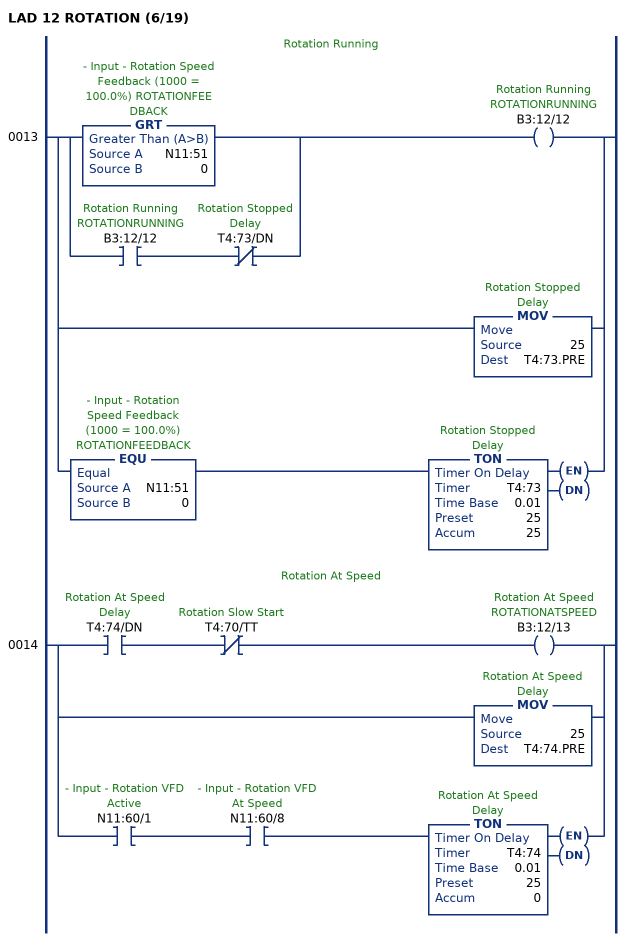
% Rung: 13 %
% Rotation Running %
SOR BST BST GRT N11:51 0 NXB XIC B3:12/12 XIO T4:73/DN BND OTE B3:12/12 NXB MOV 25 T4:73.PRE NXB EQU N11:51 0 TON T4:73 0.01 25 25 BND EOR
%   N11:51  ROTATIONFEEDBACK  "- Input - Rotation Speed Feedback (1000 = 100.0%)" %
%   B3:12/12  ROTATIONRUNNING  "Rotation Running" %
%   T4:73  "Rotation Stopped Delay" %
% Rung: 14 %
% Rotation At Speed %
SOR BST XIC T4:74/DN XIO T4:70/TT OTE B3:12/13 NXB MOV 25 T4:74.PRE NXB XIC N11:60/1 XIC N11:60/8 TON T4:74 0.01 25 0 BND EOR
%   T4:74  "Rotation At Speed Delay" %
%   T4:70  "Rotation Slow Start" %
%   B3:12/13  ROTATIONATSPEED  "Rotation At Speed" %
%   N11:60/1  "- Input - Rotation VFD Active" %
%   N11:60/8  "- Input - Rotation VFD At Speed" %

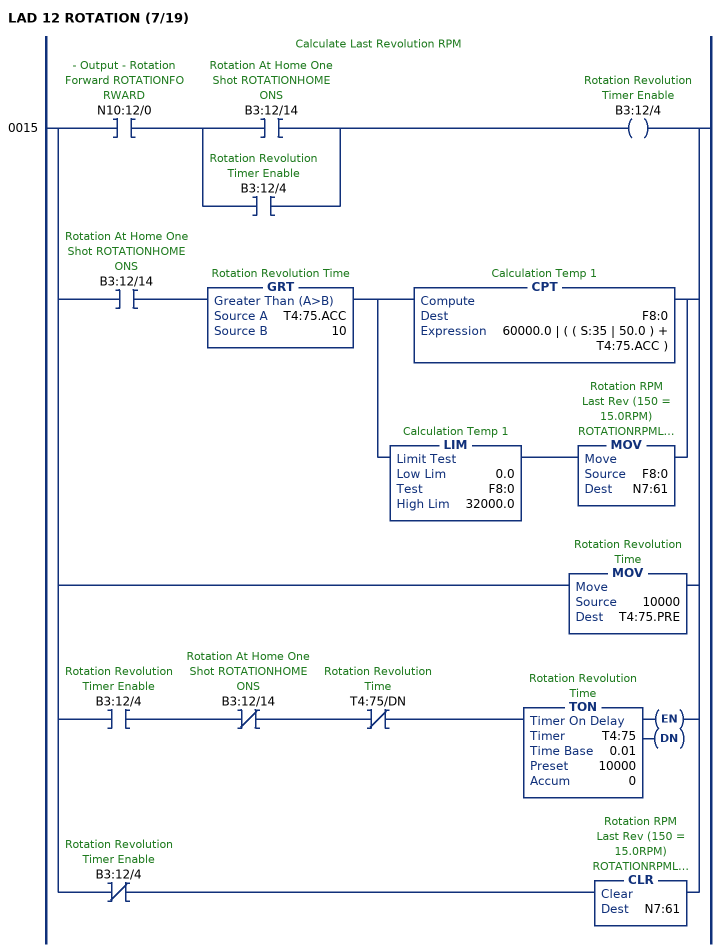
% Rung: 15 %
% Calculate Last Revolution RPM %
SOR BST XIC N10:12/0 BST XIC B3:12/14 NXB XIC B3:12/4 BND OTE B3:12/4 NXB XIC B3:12/14 GRT T4:75.ACC 10 BST CPT F8:0 " 60000.0 | ( ( S:35 | 50.0 ) + T4:75.ACC ) " NXB LIM 0.0 F8:0 32000.0 MOV F8:0 N7:61 BND NXB MOV 10000 T4:75.PRE NXB XIC B3:12/4 XIO B3:12/14 XIO T4:75/DN TON T4:75 0.01 10000 0 NXB XIO B3:12/4 CLR N7:61 BND EOR
%   N10:12/0  ROTATIONFORWARD  "- Output - Rotation Forward" %
%   B3:12/14  ROTATIONHOMEONS  "Rotation At Home One Shot" %
%   B3:12/4  "Rotation Revolution Timer Enable" %
%   T4:75  "Rotation Revolution Time" %
%   F8:0  "Calculation Temp 1" %
%   S:35  "Last 1 ms Scan Time" %
%   N7:61  ROTATIONRPMLAST  "Rotation RPM Last Rev (150 = 15.0RPM)" %

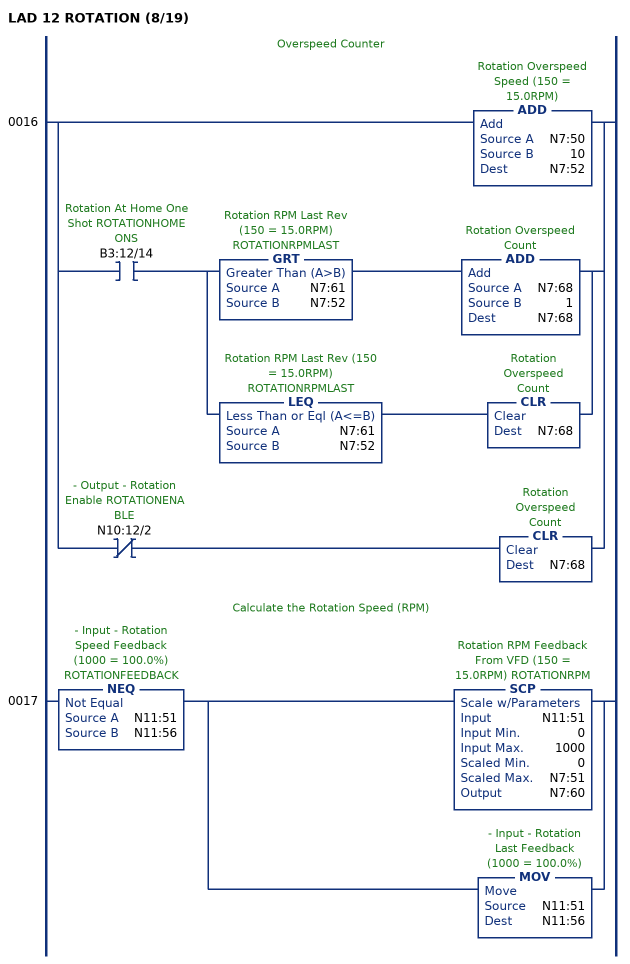
% Rung: 16 %
% Overspeed Counter %
SOR BST ADD N7:50 10 N7:52 NXB XIC B3:12/14 BST GRT N7:61 N7:52 ADD N7:68 1 N7:68 NXB LEQ N7:61 N7:52 CLR N7:68 BND NXB XIO N10:12/2 CLR N7:68 BND EOR
%   N7:50  ROTATIONBASESPEED  "Rotation Base Speed (150 = 15.0RPM)" %
%   N7:52  "Rotation Overspeed Speed (150 = 15.0RPM)" %
%   B3:12/14  ROTATIONHOMEONS  "Rotation At Home One Shot" %
%   N7:61  ROTATIONRPMLAST  "Rotation RPM Last Rev (150 = 15.0RPM)" %
%   N7:68  "Rotation Overspeed Count" %
%   N10:12/2  ROTATIONENABLE  "- Output - Rotation Enable" %
% Rung: 17 %
% Calculate the Rotation Speed (RPM) %
SOR NEQ N11:51 N11:56 BST SCP N11:51 0 1000 0 N7:51 N7:60 NXB MOV N11:51 N11:56 BND EOR
%   N11:51  ROTATIONFEEDBACK  "- Input - Rotation Speed Feedback (1000 = 100.0%)" %
%   N11:56  "- Input - Rotation Last Feedback (1000 = 100.0%)" %
%   N7:51  ROTATIONMAXSPEED  "Rotation Max Speed (150 = 15.0RPM)" %
%   N7:60  ROTATIONRPM  "Rotation RPM Feedback From VFD (150 = 15.0RPM)" %

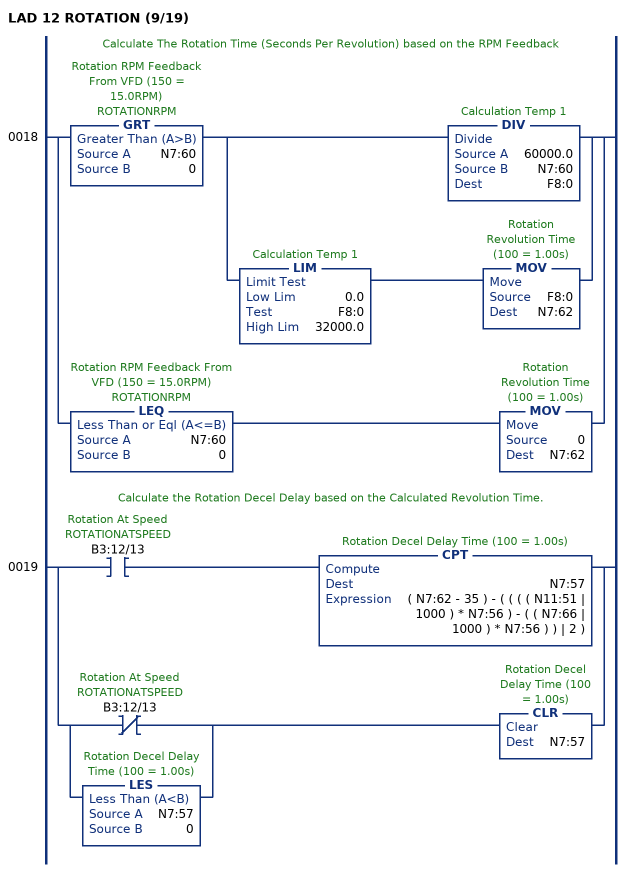
% Rung: 18 %
% Calculate The Rotation Time (Seconds Per Revolution) based on the RPM Feedback %
SOR BST GRT N7:60 0 BST DIV 60000.0 N7:60 F8:0 NXB LIM 0.0 F8:0 32000.0 MOV F8:0 N7:62 BND NXB LEQ N7:60 0 MOV 0 N7:62 BND EOR
%   N7:60  ROTATIONRPM  "Rotation RPM Feedback From VFD (150 = 15.0RPM)" %
%   F8:0  "Calculation Temp 1" %
%   N7:62  "Rotation Revolution Time (100 = 1.00s)" %
% Rung: 19 %
% Calculate the Rotation Decel Delay based on the Calculated Revolution Time. %
SOR BST XIC B3:12/13 CPT N7:57 " ( N7:62 - 35 ) - ( ( ( ( N11:51 | 1000 ) * N7:56 ) - ( ( N7:66 | 1000 ) * N7:56 ) ) | 2 ) " NXB BST XIO B3:12/13 NXB LES N7:57 0 BND CLR N7:57 BND EOR
%   B3:12/13  ROTATIONATSPEED  "Rotation At Speed" %
%   N7:57  "Rotation Decel Delay Time (100 = 1.00s)" %
%   N7:62  "Rotation Revolution Time (100 = 1.00s)" %
%   N11:51  ROTATIONFEEDBACK  "- Input - Rotation Speed Feedback (1000 = 100.0%)" %
%   N7:56  "Rotation Decel Time (100 = 1.00s)" %
%   N7:66  "Rotation Home Speed (25 = 2.5RPM)" %

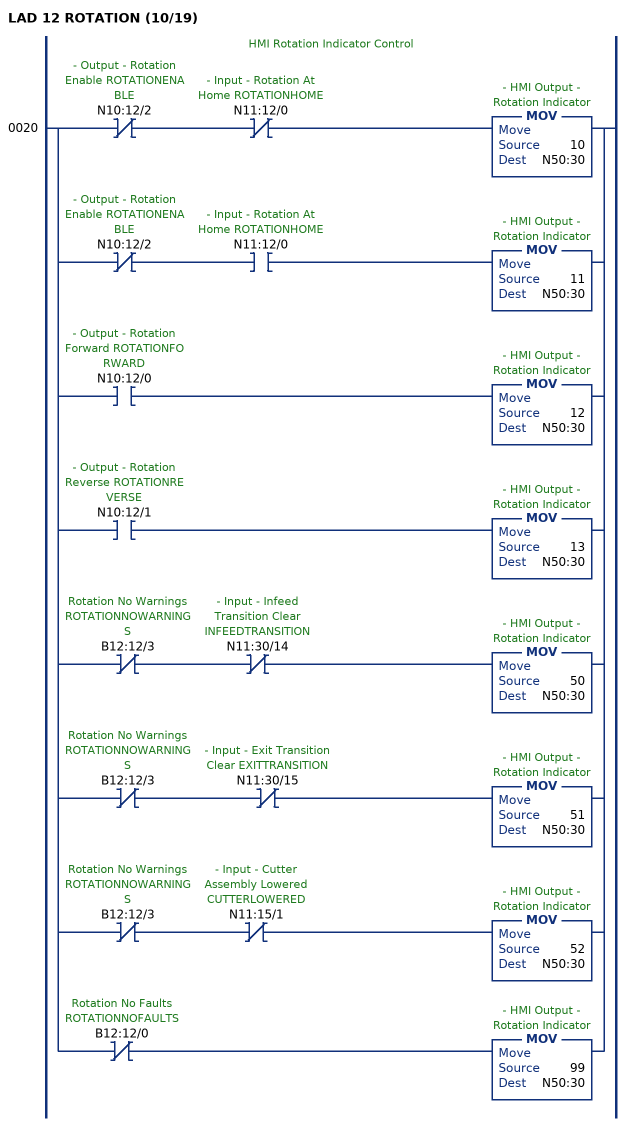
% Rung: 20 %
% HMI Rotation Indicator Control %
SOR BST XIO N10:12/2 XIO N11:12/0 MOV 10 N50:30 NXB XIO N10:12/2 XIC N11:12/0 MOV 11 N50:30 NXB XIC N10:12/0 MOV 12 N50:30 NXB XIC N10:12/1 MOV 13 N50:30 NXB XIO B12:12/3 XIO N11:30/14 MOV 50 N50:30 NXB XIO B12:12/3 XIO N11:30/15 MOV 51 N50:30 NXB XIO B12:12/3 XIO N11:15/1 MOV 52 N50:30 NXB XIO B12:12/0 MOV 99 N50:30 BND EOR
%   N10:12/2  ROTATIONENABLE  "- Output - Rotation Enable" %
%   N11:12/0  ROTATIONHOME  "- Input - Rotation At Home" %
%   N50:30  "- HMI Output - Rotation Indicator" %
%   N10:12/0  ROTATIONFORWARD  "- Output - Rotation Forward" %
%   N10:12/1  ROTATIONREVERSE  "- Output - Rotation Reverse" %
%   B12:12/3  ROTATIONNOWARNINGS  "Rotation No Warnings" %
%   N11:30/14  INFEEDTRANSITION  "- Input - Infeed Transition Clear" %
%   N11:30/15  EXITTRANSITION  "- Input - Exit Transition Clear" %
%   N11:15/1  CUTTERLOWERED  "- Input - Cutter Assembly Lowered" %
%   B12:12/0  ROTATIONNOFAULTS  "Rotation No Faults" %

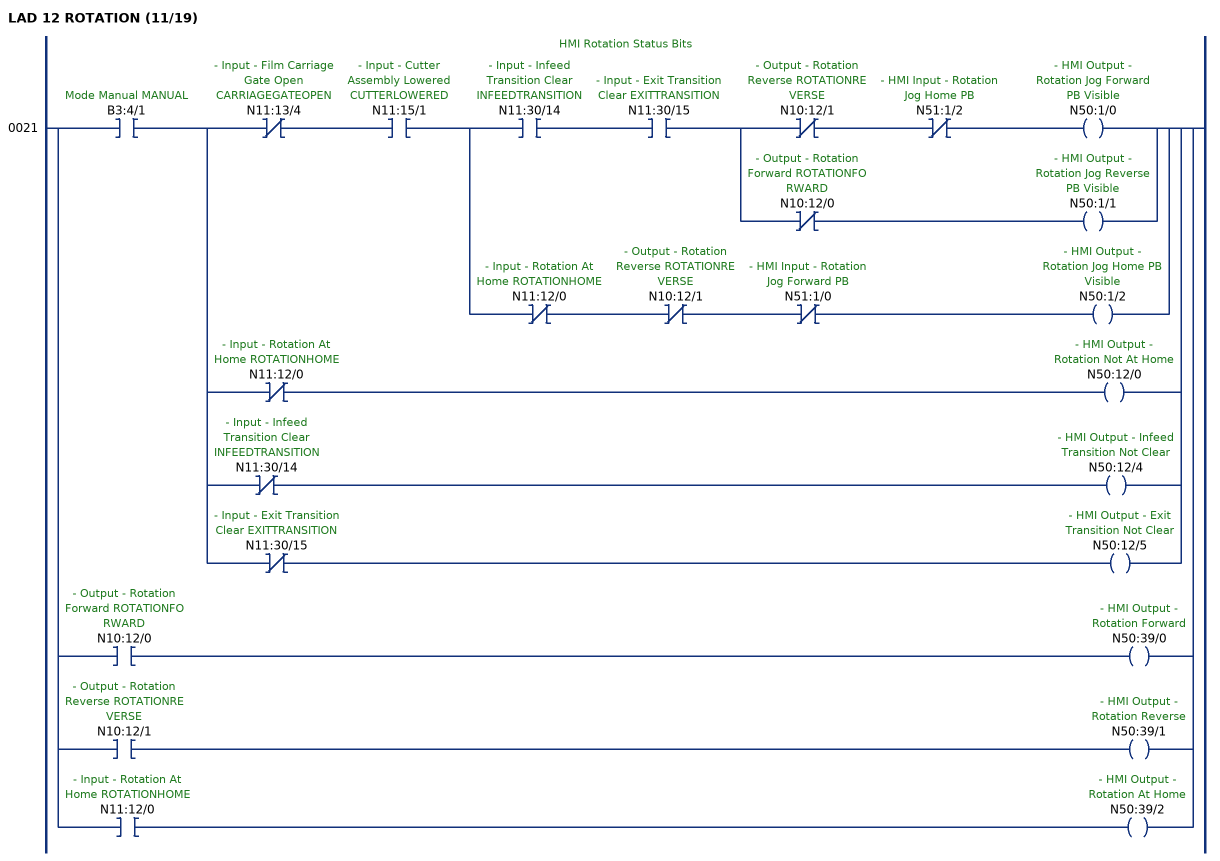
% Rung: 21 %
% HMI Rotation Status Bits %
SOR BST XIC B3:4/1 BST XIO N11:13/4 XIC N11:15/1 BST XIC N11:30/14 XIC N11:30/15 BST XIO N10:12/1 XIO N51:1/2 OTE N50:1/0 NXB XIO N10:12/0 OTE N50:1/1 BND NXB XIO N11:12/0 XIO N10:12/1 XIO N51:1/0 OTE N50:1/2 BND NXB XIO N11:12/0 OTE N50:12/0 NXB XIO N11:30/14 OTE N50:12/4 NXB XIO N11:30/15 OTE N50:12/5 BND NXB XIC N10:12/0 OTE N50:39/0 NXB XIC N10:12/1 OTE N50:39/1 NXB XIC N11:12/0 OTE N50:39/2 BND EOR
%   B3:4/1  MANUAL  "Mode Manual" %
%   N11:13/4  CARRIAGEGATEOPEN  "- Input - Film Carriage Gate Open" %
%   N11:15/1  CUTTERLOWERED  "- Input - Cutter Assembly Lowered" %
%   N11:30/14  INFEEDTRANSITION  "- Input - Infeed Transition Clear" %
%   N11:30/15  EXITTRANSITION  "- Input - Exit Transition Clear" %
%   N10:12/1  ROTATIONREVERSE  "- Output - Rotation Reverse" %
%   N51:1/2  "- HMI Input - Rotation Jog Home PB" %
%   N50:1/0  "- HMI Output - Rotation Jog Forward PB Visible" %
%   N10:12/0  ROTATIONFORWARD  "- Output - Rotation Forward" %
%   N50:1/1  "- HMI Output - Rotation Jog Reverse PB Visible" %
%   N11:12/0  ROTATIONHOME  "- Input - Rotation At Home" %
%   N51:1/0  "- HMI Input - Rotation Jog Forward PB" %
%   N50:1/2  "- HMI Output - Rotation Jog Home PB Visible" %
%   N50:12/0  "- HMI Output - Rotation Not At Home" %
%   N50:12/4  "- HMI Output - Infeed Transition Not Clear" %
%   N50:12/5  "- HMI Output - Exit Transition Not Clear" %
%   N50:39/0  "- HMI Output - Rotation Forward" %
%   N50:39/1  "- HMI Output - Rotation Reverse" %
%   N50:39/2  "- HMI Output - Rotation At Home" %

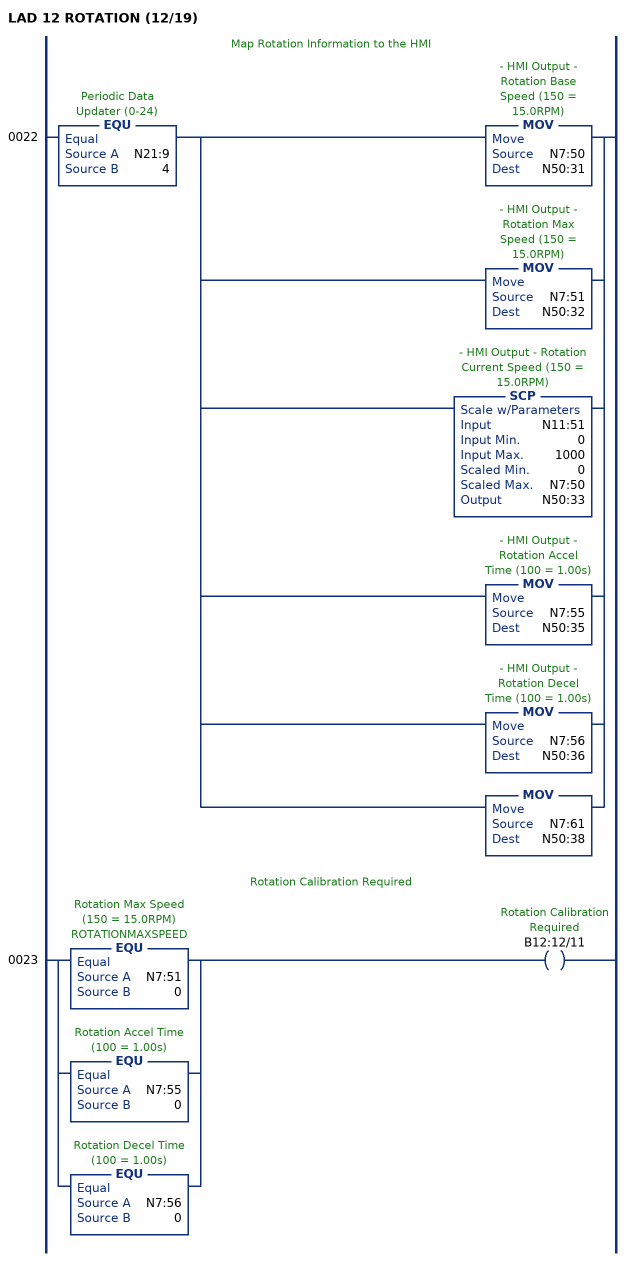
% Rung: 22 %
% Map Rotation Information to the HMI %
SOR EQU N21:9 4 BST MOV N7:50 N50:31 NXB MOV N7:51 N50:32 NXB SCP N11:51 0 1000 0 N7:50 N50:33 NXB MOV N7:55 N50:35 NXB MOV N7:56 N50:36 NXB MOV N7:61 N50:38 BND EOR
%   N21:9  "Periodic Data Updater (0-24)" %
%   N7:50  ROTATIONBASESPEED  "Rotation Base Speed (150 = 15.0RPM)" %
%   N50:31  "- HMI Output - Rotation Base Speed (150 = 15.0RPM)" %
%   N7:51  ROTATIONMAXSPEED  "Rotation Max Speed (150 = 15.0RPM)" %
%   N50:32  "- HMI Output - Rotation Max Speed (150 = 15.0RPM)" %
%   N11:51  ROTATIONFEEDBACK  "- Input - Rotation Speed Feedback (1000 = 100.0%)" %
%   N50:33  "- HMI Output - Rotation Current Speed (150 = 15.0RPM)" %
%   N7:55  "Rotation Accel Time (100 = 1.00s)" %
%   N50:35  "- HMI Output - Rotation Accel Time (100 = 1.00s)" %
%   N7:56  "Rotation Decel Time (100 = 1.00s)" %
%   N50:36  "- HMI Output - Rotation Decel Time (100 = 1.00s)" %
%   N7:61  ROTATIONRPMLAST  "Rotation RPM Last Rev (150 = 15.0RPM)" %
% Rung: 23 %
% Rotation Calibration Required %
SOR BST EQU N7:51 0 NXB EQU N7:55 0 NXB EQU N7:56 0 BND OTE B12:12/11 EOR
%   N7:51  ROTATIONMAXSPEED  "Rotation Max Speed (150 = 15.0RPM)" %
%   N7:55  "Rotation Accel Time (100 = 1.00s)" %
%   N7:56  "Rotation Decel Time (100 = 1.00s)" %
%   B12:12/11  "Rotation Calibration Required" %

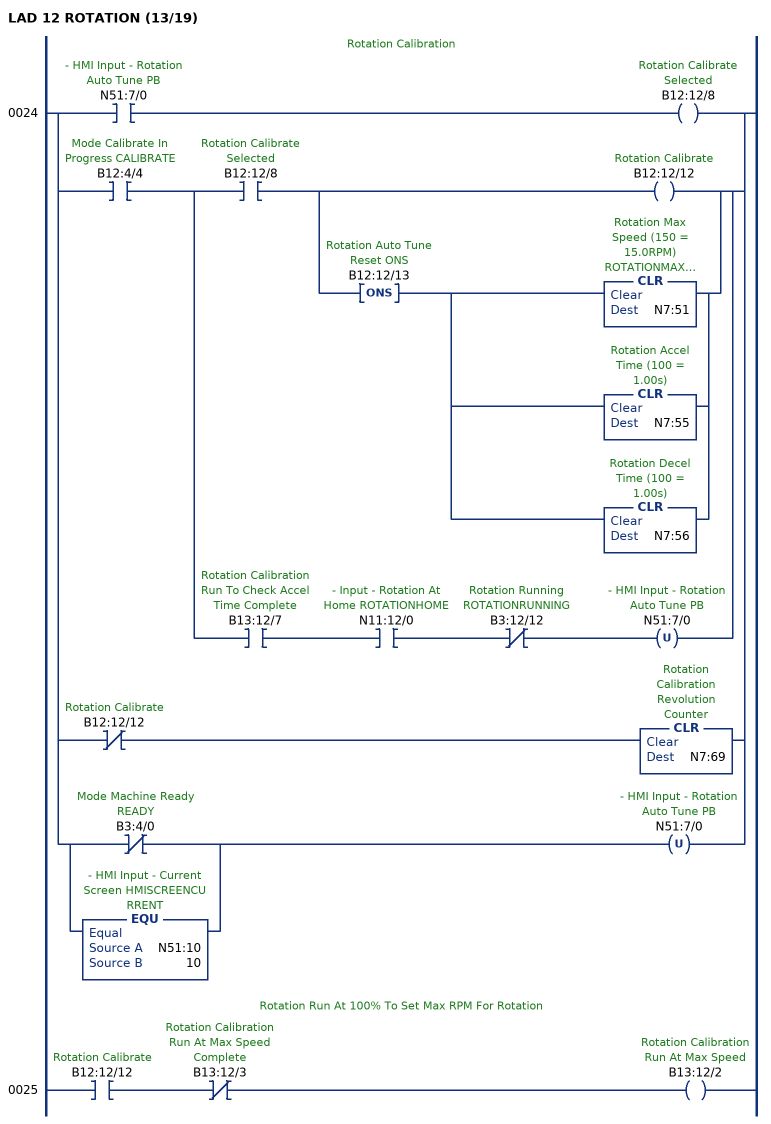
% Rung: 24 %
% Rotation Calibration %
SOR BST XIC N51:7/0 OTE B12:12/8 NXB XIC B12:4/4 BST XIC B12:12/8 BST OTE B12:12/12 NXB ONS B12:12/13 BST CLR N7:51 NXB CLR N7:55 NXB CLR N7:56 BND BND NXB XIC B13:12/7 XIC N11:12/0 XIO B3:12/12 OTU N51:7/0 BND NXB XIO B12:12/12 CLR N7:69 NXB BST XIO B3:4/0 NXB EQU N51:10 10 BND OTU N51:7/0 BND EOR
%   N51:7/0  "- HMI Input - Rotation Auto Tune PB" %
%   B12:12/8  "Rotation Calibrate Selected" %
%   B12:4/4  CALIBRATE  "Mode Calibrate In Progress" %
%   B12:12/12  "Rotation Calibrate" %
%   B12:12/13  "Rotation Auto Tune Reset ONS" %
%   N7:51  ROTATIONMAXSPEED  "Rotation Max Speed (150 = 15.0RPM)" %
%   N7:55  "Rotation Accel Time (100 = 1.00s)" %
%   N7:56  "Rotation Decel Time (100 = 1.00s)" %
%   B13:12/7  "Rotation Calibration Run To Check Accel Time Complete" %
%   N11:12/0  ROTATIONHOME  "- Input - Rotation At Home" %
%   B3:12/12  ROTATIONRUNNING  "Rotation Running" %
%   N7:69  "Rotation Calibration Revolution Counter" %
%   B3:4/0  READY  "Mode Machine Ready" %
%   N51:10  HMISCREENCURRENT  "- HMI Input - Current Screen" %
% Rung: 25 %
% Rotation Run At 100% To Set Max RPM For Rotation %
SOR XIC B12:12/12 XIO B13:12/3 OTE B13:12/2 EOR
%   B12:12/12  "Rotation Calibrate" %
%   B13:12/3  "Rotation Calibration Run At Max Speed Complete" %
%   B13:12/2  "Rotation Calibration Run At Max Speed" %

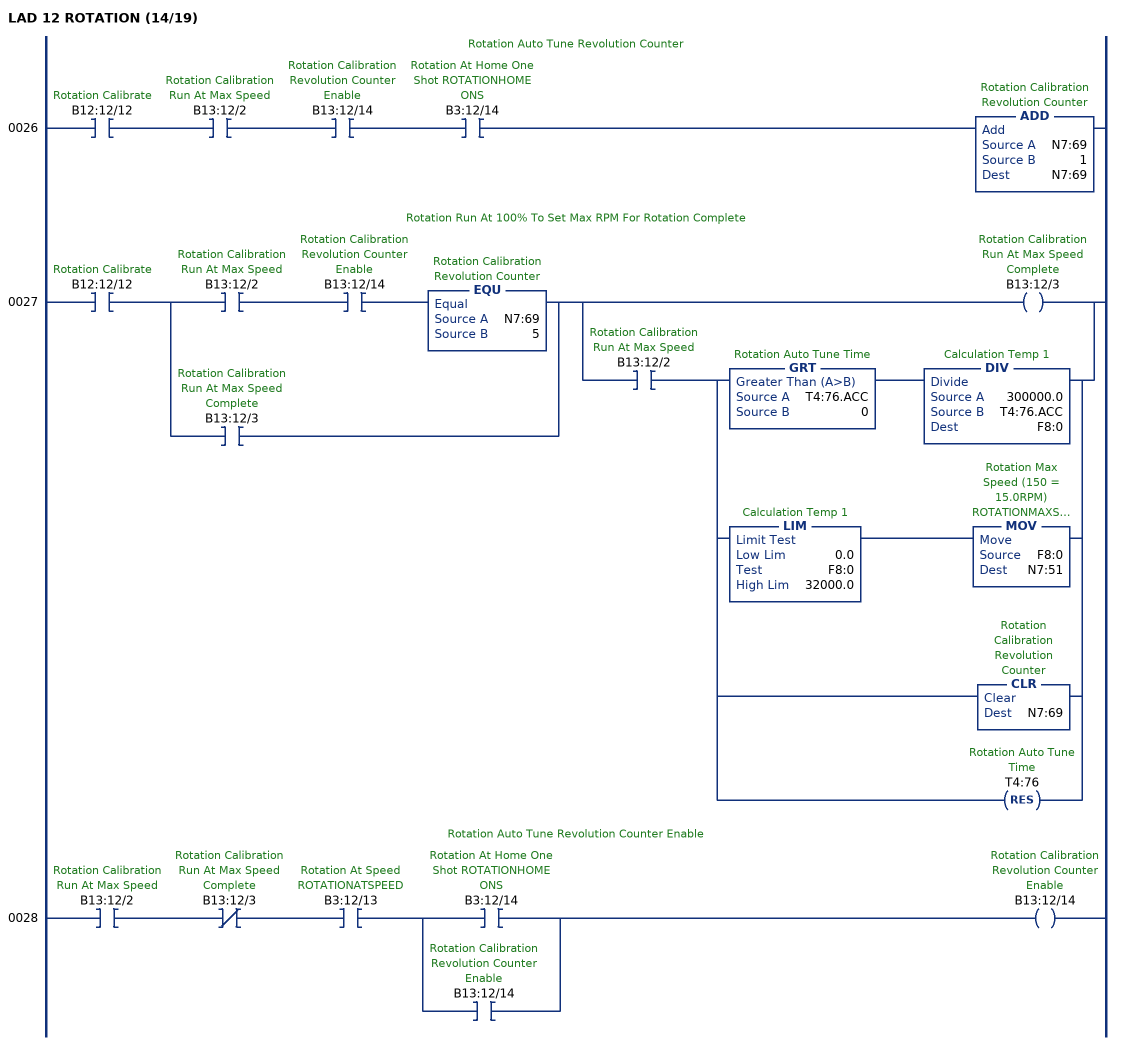
% Rung: 26 %
% Rotation Auto Tune Revolution Counter %
SOR XIC B12:12/12 XIC B13:12/2 XIC B13:12/14 XIC B3:12/14 ADD N7:69 1 N7:69 EOR
%   B12:12/12  "Rotation Calibrate" %
%   B13:12/2  "Rotation Calibration Run At Max Speed" %
%   B13:12/14  "Rotation Calibration Revolution Counter Enable" %
%   B3:12/14  ROTATIONHOMEONS  "Rotation At Home One Shot" %
%   N7:69  "Rotation Calibration Revolution Counter" %
% Rung: 27 %
% Rotation Run At 100% To Set Max RPM For Rotation Complete %
SOR XIC B12:12/12 BST XIC B13:12/2 XIC B13:12/14 EQU N7:69 5 NXB XIC B13:12/3 BND BST OTE B13:12/3 NXB XIC B13:12/2 BST GRT T4:76.ACC 0 DIV 300000.0 T4:76.ACC F8:0 NXB LIM 0.0 F8:0 32000.0 MOV F8:0 N7:51 NXB CLR N7:69 NXB RES T4:76 BND BND EOR
%   B12:12/12  "Rotation Calibrate" %
%   B13:12/2  "Rotation Calibration Run At Max Speed" %
%   B13:12/14  "Rotation Calibration Revolution Counter Enable" %
%   N7:69  "Rotation Calibration Revolution Counter" %
%   B13:12/3  "Rotation Calibration Run At Max Speed Complete" %
%   T4:76  "Rotation Auto Tune Time" %
%   F8:0  "Calculation Temp 1" %
%   N7:51  ROTATIONMAXSPEED  "Rotation Max Speed (150 = 15.0RPM)" %
% Rung: 28 %
% Rotation Auto Tune Revolution Counter Enable %
SOR XIC B13:12/2 XIO B13:12/3 XIC B3:12/13 BST XIC B3:12/14 NXB XIC B13:12/14 BND OTE B13:12/14 EOR
%   B13:12/2  "Rotation Calibration Run At Max Speed" %
%   B13:12/3  "Rotation Calibration Run At Max Speed Complete" %
%   B3:12/13  ROTATIONATSPEED  "Rotation At Speed" %
%   B3:12/14  ROTATIONHOMEONS  "Rotation At Home One Shot" %
%   B13:12/14  "Rotation Calibration Revolution Counter Enable" %

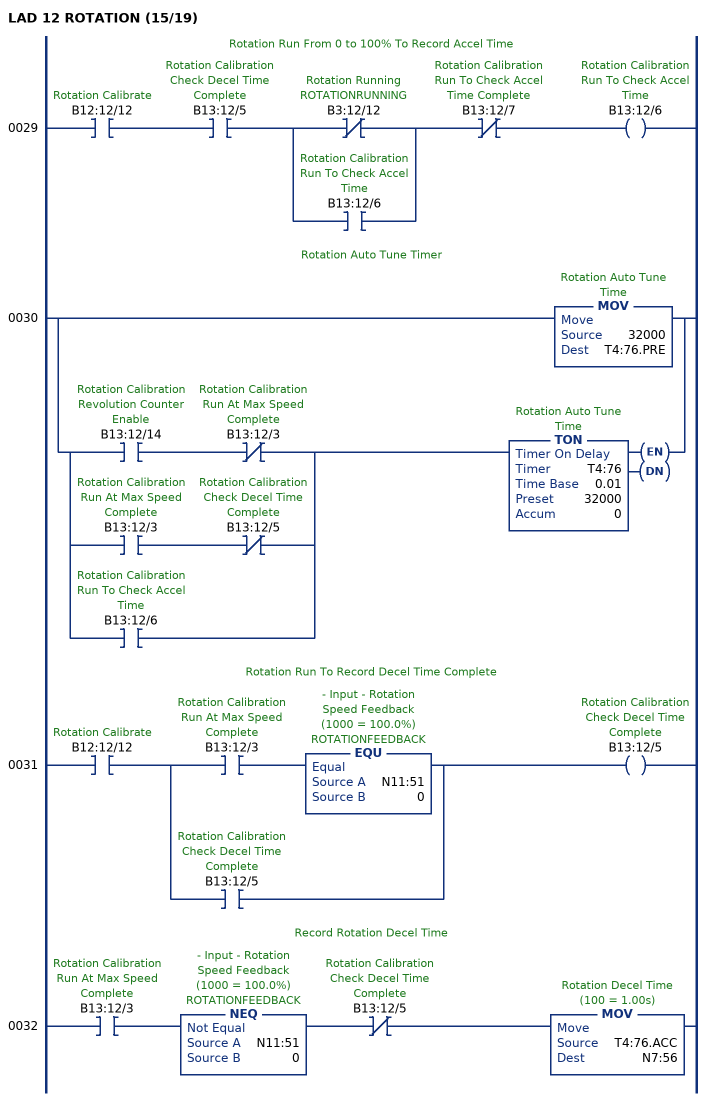
% Rung: 29 %
% Rotation Run From 0 to 100% To Record Accel Time %
SOR XIC B12:12/12 XIC B13:12/5 BST XIO B3:12/12 NXB XIC B13:12/6 BND XIO B13:12/7 OTE B13:12/6 EOR
%   B12:12/12  "Rotation Calibrate" %
%   B13:12/5  "Rotation Calibration Check Decel Time Complete" %
%   B3:12/12  ROTATIONRUNNING  "Rotation Running" %
%   B13:12/6  "Rotation Calibration Run To Check Accel Time" %
%   B13:12/7  "Rotation Calibration Run To Check Accel Time Complete" %
% Rung: 30 %
% Rotation Auto Tune Timer %
SOR BST MOV 32000 T4:76.PRE NXB BST XIC B13:12/14 XIO B13:12/3 NXB XIC B13:12/3 XIO B13:12/5 NXB XIC B13:12/6 BND TON T4:76 0.01 32000 0 BND EOR
%   T4:76  "Rotation Auto Tune Time" %
%   B13:12/14  "Rotation Calibration Revolution Counter Enable" %
%   B13:12/3  "Rotation Calibration Run At Max Speed Complete" %
%   B13:12/5  "Rotation Calibration Check Decel Time Complete" %
%   B13:12/6  "Rotation Calibration Run To Check Accel Time" %
% Rung: 31 %
% Rotation Run To Record Decel Time Complete %
SOR XIC B12:12/12 BST XIC B13:12/3 EQU N11:51 0 NXB XIC B13:12/5 BND OTE B13:12/5 EOR
%   B12:12/12  "Rotation Calibrate" %
%   B13:12/3  "Rotation Calibration Run At Max Speed Complete" %
%   N11:51  ROTATIONFEEDBACK  "- Input - Rotation Speed Feedback (1000 = 100.0%)" %
%   B13:12/5  "Rotation Calibration Check Decel Time Complete" %
% Rung: 32 %
% Record Rotation Decel Time %
SOR XIC B13:12/3 NEQ N11:51 0 XIO B13:12/5 MOV T4:76.ACC N7:56 EOR
%   B13:12/3  "Rotation Calibration Run At Max Speed Complete" %
%   N11:51  ROTATIONFEEDBACK  "- Input - Rotation Speed Feedback (1000 = 100.0%)" %
%   B13:12/5  "Rotation Calibration Check Decel Time Complete" %
%   T4:76  "Rotation Auto Tune Time" %
%   N7:56  "Rotation Decel Time (100 = 1.00s)" %

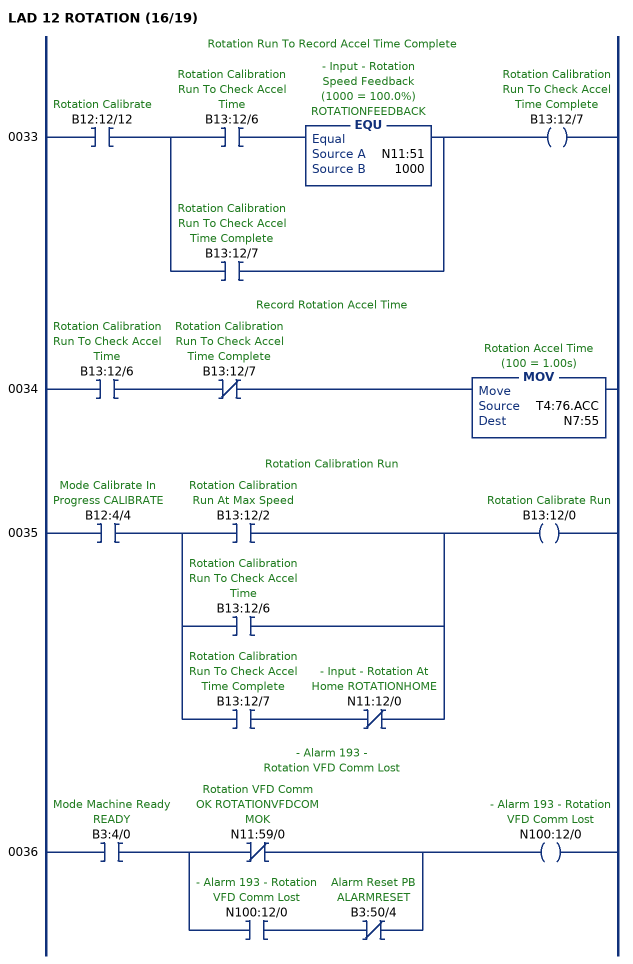
% Rung: 33 %
% Rotation Run To Record Accel Time Complete %
SOR XIC B12:12/12 BST XIC B13:12/6 EQU N11:51 1000 NXB XIC B13:12/7 BND OTE B13:12/7 EOR
%   B12:12/12  "Rotation Calibrate" %
%   B13:12/6  "Rotation Calibration Run To Check Accel Time" %
%   N11:51  ROTATIONFEEDBACK  "- Input - Rotation Speed Feedback (1000 = 100.0%)" %
%   B13:12/7  "Rotation Calibration Run To Check Accel Time Complete" %
% Rung: 34 %
% Record Rotation Accel Time %
SOR XIC B13:12/6 XIO B13:12/7 MOV T4:76.ACC N7:55 EOR
%   B13:12/6  "Rotation Calibration Run To Check Accel Time" %
%   B13:12/7  "Rotation Calibration Run To Check Accel Time Complete" %
%   T4:76  "Rotation Auto Tune Time" %
%   N7:55  "Rotation Accel Time (100 = 1.00s)" %
% Rung: 35 %
% Rotation Calibration Run %
SOR XIC B12:4/4 BST XIC B13:12/2 NXB XIC B13:12/6 NXB XIC B13:12/7 XIO N11:12/0 BND OTE B13:12/0 EOR
%   B12:4/4  CALIBRATE  "Mode Calibrate In Progress" %
%   B13:12/2  "Rotation Calibration Run At Max Speed" %
%   B13:12/6  "Rotation Calibration Run To Check Accel Time" %
%   B13:12/7  "Rotation Calibration Run To Check Accel Time Complete" %
%   N11:12/0  ROTATIONHOME  "- Input - Rotation At Home" %
%   B13:12/0  "Rotation Calibrate Run" %
% Rung: 36 %
% - Alarm 193 -
% 
% Rotation VFD Comm Lost %
SOR XIC B3:4/0 BST XIO N11:59/0 NXB XIC N100:12/0 XIO B3:50/4 BND OTE N100:12/0 EOR
%   B3:4/0  READY  "Mode Machine Ready" %
%   N11:59/0  ROTATIONVFDCOMMOK  "Rotation VFD Comm OK" %
%   N100:12/0  "- Alarm 193 - Rotation VFD Comm Lost" %
%   B3:50/4  ALARMRESET  "Alarm Reset PB" %

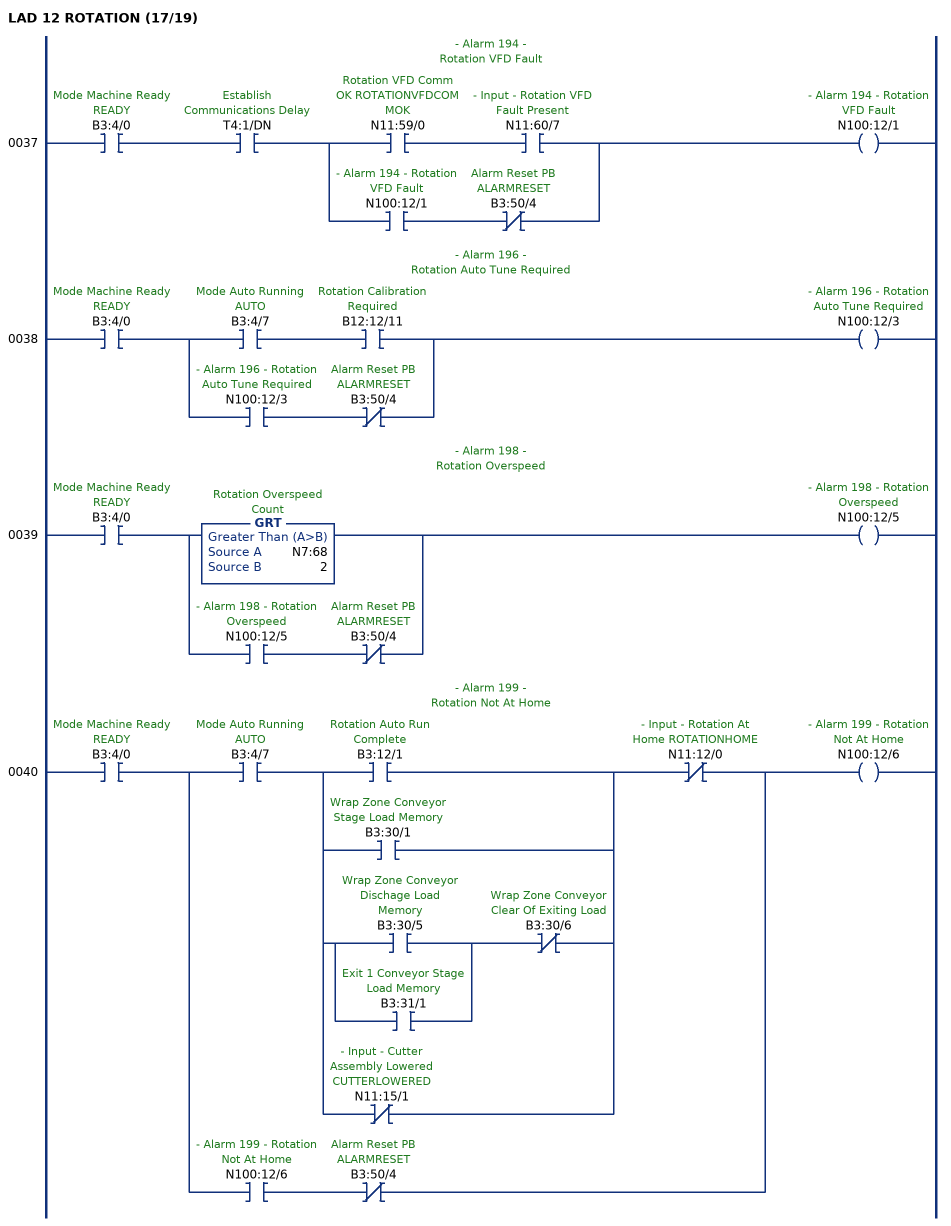
% Rung: 37 %
% - Alarm 194 -
% 
% Rotation VFD Fault %
SOR XIC B3:4/0 XIC T4:1/DN BST XIC N11:59/0 XIC N11:60/7 NXB XIC N100:12/1 XIO B3:50/4 BND OTE N100:12/1 EOR
%   B3:4/0  READY  "Mode Machine Ready" %
%   T4:1  "Establish Communications Delay" %
%   N11:59/0  ROTATIONVFDCOMMOK  "Rotation VFD Comm OK" %
%   N11:60/7  "- Input - Rotation VFD Fault Present" %
%   N100:12/1  "- Alarm 194 - Rotation VFD Fault" %
%   B3:50/4  ALARMRESET  "Alarm Reset PB" %
% Rung: 38 %
% - Alarm 196 -
% 
% Rotation Auto Tune Required %
SOR XIC B3:4/0 BST XIC B3:4/7 XIC B12:12/11 NXB XIC N100:12/3 XIO B3:50/4 BND OTE N100:12/3 EOR
%   B3:4/0  READY  "Mode Machine Ready" %
%   B3:4/7  AUTO  "Mode Auto Running" %
%   B12:12/11  "Rotation Calibration Required" %
%   N100:12/3  "- Alarm 196 - Rotation Auto Tune Required" %
%   B3:50/4  ALARMRESET  "Alarm Reset PB" %
% Rung: 39 %
% - Alarm 198 -
% 
% Rotation Overspeed %
SOR XIC B3:4/0 BST GRT N7:68 2 NXB XIC N100:12/5 XIO B3:50/4 BND OTE N100:12/5 EOR
%   B3:4/0  READY  "Mode Machine Ready" %
%   N7:68  "Rotation Overspeed Count" %
%   N100:12/5  "- Alarm 198 - Rotation Overspeed" %
%   B3:50/4  ALARMRESET  "Alarm Reset PB" %
% Rung: 40 %
% - Alarm 199 -
% 
% Rotation Not At Home %
SOR XIC B3:4/0 BST XIC B3:4/7 BST XIC B3:12/1 NXB XIC B3:30/1 NXB BST XIC B3:30/5 NXB XIC B3:31/1 BND XIO B3:30/6 NXB XIO N11:15/1 BND XIO N11:12/0 NXB XIC N100:12/6 XIO B3:50/4 BND OTE N100:12/6 EOR
%   B3:4/0  READY  "Mode Machine Ready" %
%   B3:4/7  AUTO  "Mode Auto Running" %
%   B3:12/1  "Rotation Auto Run Complete" %
%   B3:30/1  "Wrap Zone Conveyor Stage Load Memory" %
%   B3:30/5  "Wrap Zone Conveyor Dischage Load Memory" %
%   B3:31/1  "Exit 1 Conveyor Stage Load Memory" %
%   B3:30/6  "Wrap Zone Conveyor Clear Of Exiting Load" %
%   N11:15/1  CUTTERLOWERED  "- Input - Cutter Assembly Lowered" %
%   N11:12/0  ROTATIONHOME  "- Input - Rotation At Home" %
%   N100:12/6  "- Alarm 199 - Rotation Not At Home" %
%   B3:50/4  ALARMRESET  "Alarm Reset PB" %

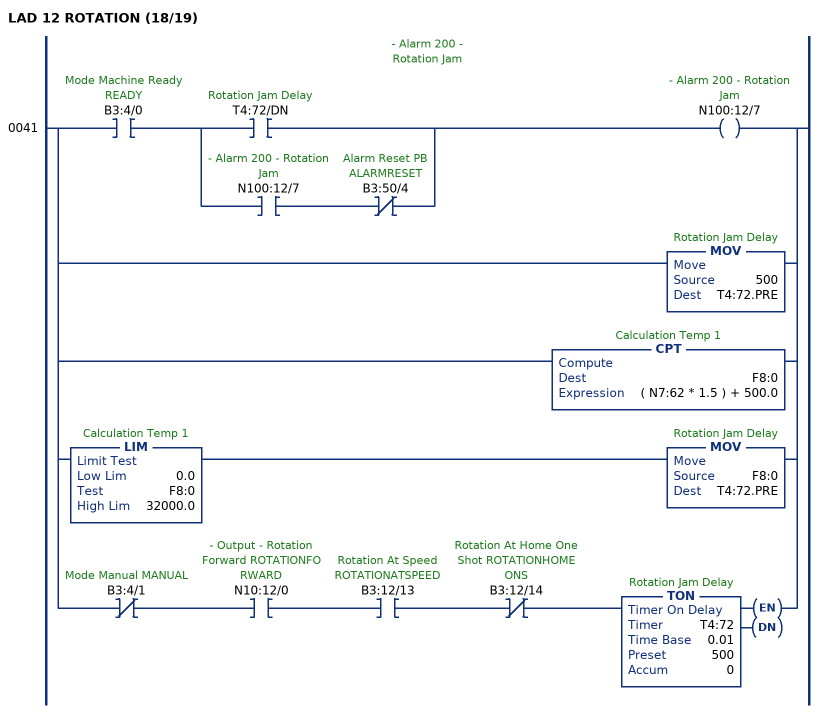
% Rung: 41 %
% - Alarm 200 -
% 
% Rotation Jam %
SOR BST XIC B3:4/0 BST XIC T4:72/DN NXB XIC N100:12/7 XIO B3:50/4 BND OTE N100:12/7 NXB BST MOV 500 T4:72.PRE NXB CPT F8:0 " ( N7:62 * 1.5 ) + 500.0 " NXB LIM 0.0 F8:0 32000.0 MOV F8:0 T4:72.PRE BND NXB XIO B3:4/1 XIC N10:12/0 XIC B3:12/13 XIO B3:12/14 TON T4:72 0.01 500 0 BND EOR
%   B3:4/0  READY  "Mode Machine Ready" %
%   T4:72  "Rotation Jam Delay" %
%   N100:12/7  "- Alarm 200 - Rotation Jam" %
%   B3:50/4  ALARMRESET  "Alarm Reset PB" %
%   F8:0  "Calculation Temp 1" %
%   N7:62  "Rotation Revolution Time (100 = 1.00s)" %
%   B3:4/1  MANUAL  "Mode Manual" %
%   N10:12/0  ROTATIONFORWARD  "- Output - Rotation Forward" %
%   B3:12/13  ROTATIONATSPEED  "Rotation At Speed" %
%   B3:12/14  ROTATIONHOMEONS  "Rotation At Home One Shot" %

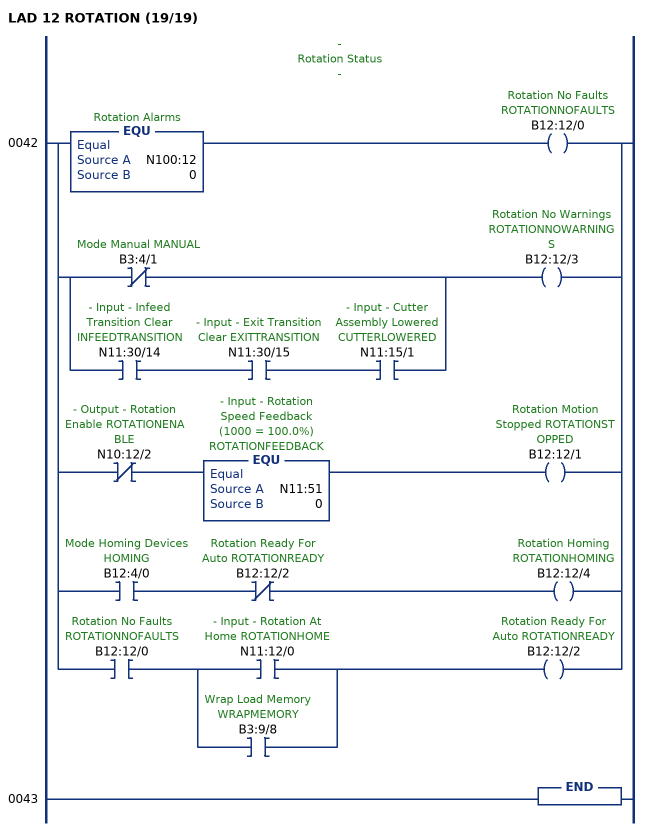
% Rung: 42 %
% -
% 
% Rotation Status
% 
% - %
SOR BST EQU N100:12 0 OTE B12:12/0 NXB BST XIO B3:4/1 NXB XIC N11:30/14 XIC N11:30/15 XIC N11:15/1 BND OTE B12:12/3 NXB XIO N10:12/2 EQU N11:51 0 OTE B12:12/1 NXB XIC B12:4/0 XIO B12:12/2 OTE B12:12/4 NXB XIC B12:12/0 BST XIC N11:12/0 NXB XIC B3:9/8 BND OTE B12:12/2 BND EOR
%   N100:12  "Rotation Alarms" %
%   B12:12/0  ROTATIONNOFAULTS  "Rotation No Faults" %
%   B3:4/1  MANUAL  "Mode Manual" %
%   N11:30/14  INFEEDTRANSITION  "- Input - Infeed Transition Clear" %
%   N11:30/15  EXITTRANSITION  "- Input - Exit Transition Clear" %
%   N11:15/1  CUTTERLOWERED  "- Input - Cutter Assembly Lowered" %
%   B12:12/3  ROTATIONNOWARNINGS  "Rotation No Warnings" %
%   N10:12/2  ROTATIONENABLE  "- Output - Rotation Enable" %
%   N11:51  ROTATIONFEEDBACK  "- Input - Rotation Speed Feedback (1000 = 100.0%)" %
%   B12:12/1  ROTATIONSTOPPED  "Rotation Motion Stopped" %
%   B12:4/0  HOMING  "Mode Homing Devices" %
%   B12:12/2  ROTATIONREADY  "Rotation Ready For Auto" %
%   B12:12/4  ROTATIONHOMING  "Rotation Homing" %
%   N11:12/0  ROTATIONHOME  "- Input - Rotation At Home" %
%   B3:9/8  WRAPMEMORY  "Wrap Load Memory" %
% Rung: 43 %
SOR END EOR

LADDER 13 "CARRIAGE"
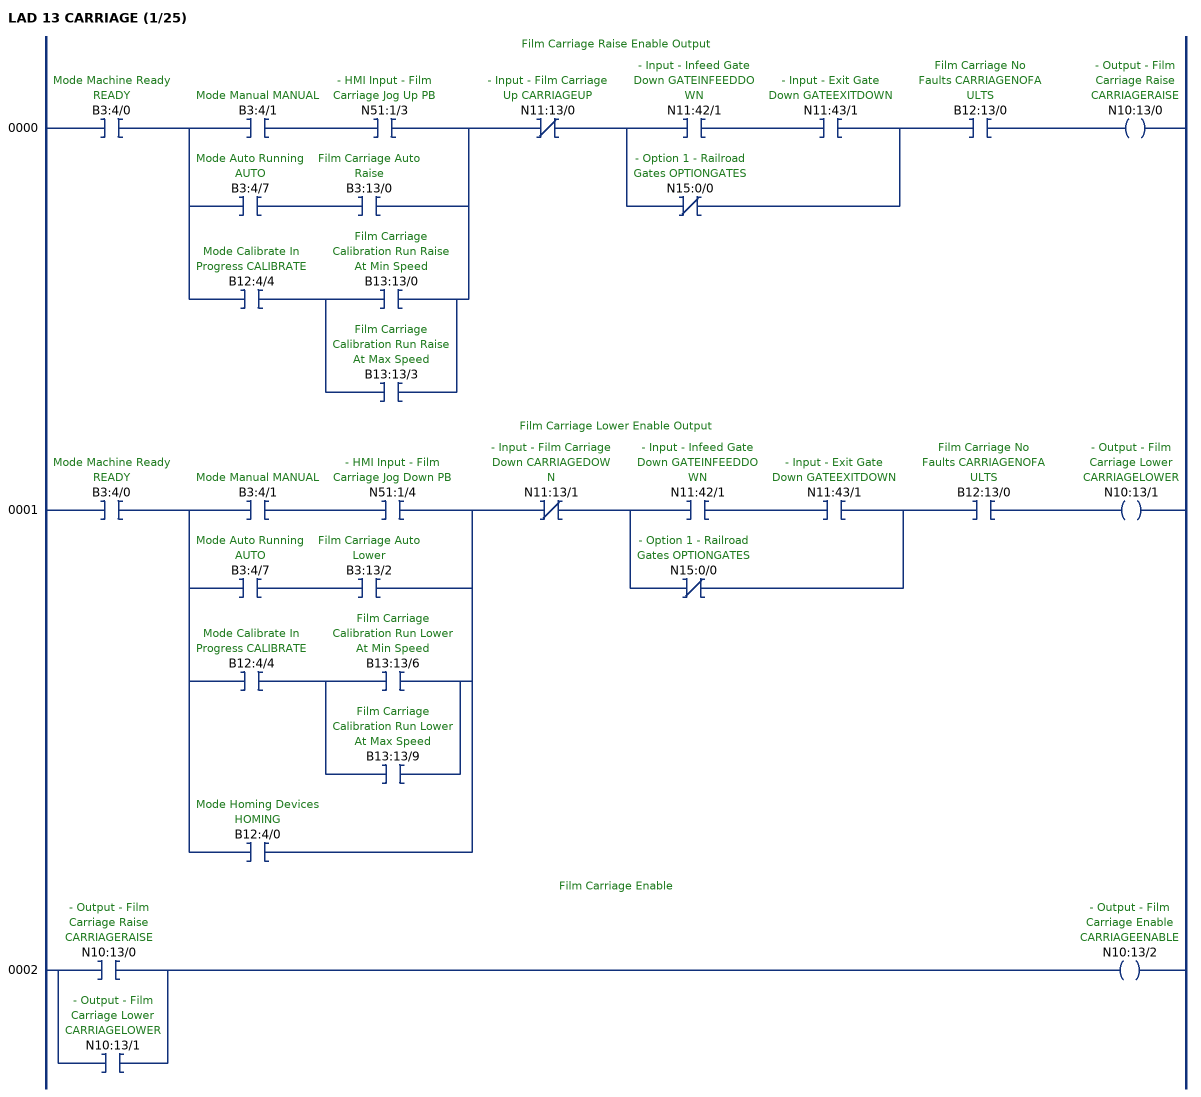
% Rung: 0 %
% Film Carriage Raise Enable Output %
SOR XIC B3:4/0 BST XIC B3:4/1 XIC N51:1/3 NXB XIC B3:4/7 XIC B3:13/0 NXB XIC B12:4/4 BST XIC B13:13/0 NXB XIC B13:13/3 BND BND XIO N11:13/0 BST XIC N11:42/1 XIC N11:43/1 NXB XIO N15:0/0 BND XIC B12:13/0 OTE N10:13/0 EOR
%   B3:4/0  READY  "Mode Machine Ready" %
%   B3:4/1  MANUAL  "Mode Manual" %
%   N51:1/3  "- HMI Input - Film Carriage Jog Up PB" %
%   B3:4/7  AUTO  "Mode Auto Running" %
%   B3:13/0  "Film Carriage Auto Raise" %
%   B12:4/4  CALIBRATE  "Mode Calibrate In Progress" %
%   B13:13/0  "Film Carriage Calibration Run Raise At Min Speed" %
%   B13:13/3  "Film Carriage Calibration Run Raise At Max Speed" %
%   N11:13/0  CARRIAGEUP  "- Input - Film Carriage Up" %
%   N11:42/1  GATEINFEEDDOWN  "- Input - Infeed Gate Down" %
%   N11:43/1  GATEEXITDOWN  "- Input - Exit Gate Down" %
%   N15:0/0  OPTIONGATES  "- Option 1 - Railroad Gates" %
%   B12:13/0  CARRIAGENOFAULTS  "Film Carriage No Faults" %
%   N10:13/0  CARRIAGERAISE  "- Output - Film Carriage Raise" %
% Rung: 1 %
% Film Carriage Lower Enable Output %
SOR XIC B3:4/0 BST XIC B3:4/1 XIC N51:1/4 NXB XIC B3:4/7 XIC B3:13/2 NXB XIC B12:4/4 BST XIC B13:13/6 NXB XIC B13:13/9 BND NXB XIC B12:4/0 BND XIO N11:13/1 BST XIC N11:42/1 XIC N11:43/1 NXB XIO N15:0/0 BND XIC B12:13/0 OTE N10:13/1 EOR
%   B3:4/0  READY  "Mode Machine Ready" %
%   B3:4/1  MANUAL  "Mode Manual" %
%   N51:1/4  "- HMI Input - Film Carriage Jog Down PB" %
%   B3:4/7  AUTO  "Mode Auto Running" %
%   B3:13/2  "Film Carriage Auto Lower" %
%   B12:4/4  CALIBRATE  "Mode Calibrate In Progress" %
%   B13:13/6  "Film Carriage Calibration Run Lower At Min Speed" %
%   B13:13/9  "Film Carriage Calibration Run Lower At Max Speed" %
%   B12:4/0  HOMING  "Mode Homing Devices" %
%   N11:13/1  CARRIAGEDOWN  "- Input - Film Carriage Down" %
%   N11:42/1  GATEINFEEDDOWN  "- Input - Infeed Gate Down" %
%   N11:43/1  GATEEXITDOWN  "- Input - Exit Gate Down" %
%   N15:0/0  OPTIONGATES  "- Option 1 - Railroad Gates" %
%   B12:13/0  CARRIAGENOFAULTS  "Film Carriage No Faults" %
%   N10:13/1  CARRIAGELOWER  "- Output - Film Carriage Lower" %
% Rung: 2 %
% Film Carriage Enable %
SOR BST XIC N10:13/0 NXB XIC N10:13/1 BND OTE N10:13/2 EOR
%   N10:13/0  CARRIAGERAISE  "- Output - Film Carriage Raise" %
%   N10:13/1  CARRIAGELOWER  "- Output - Film Carriage Lower" %
%   N10:13/2  CARRIAGEENABLE  "- Output - Film Carriage Enable" %

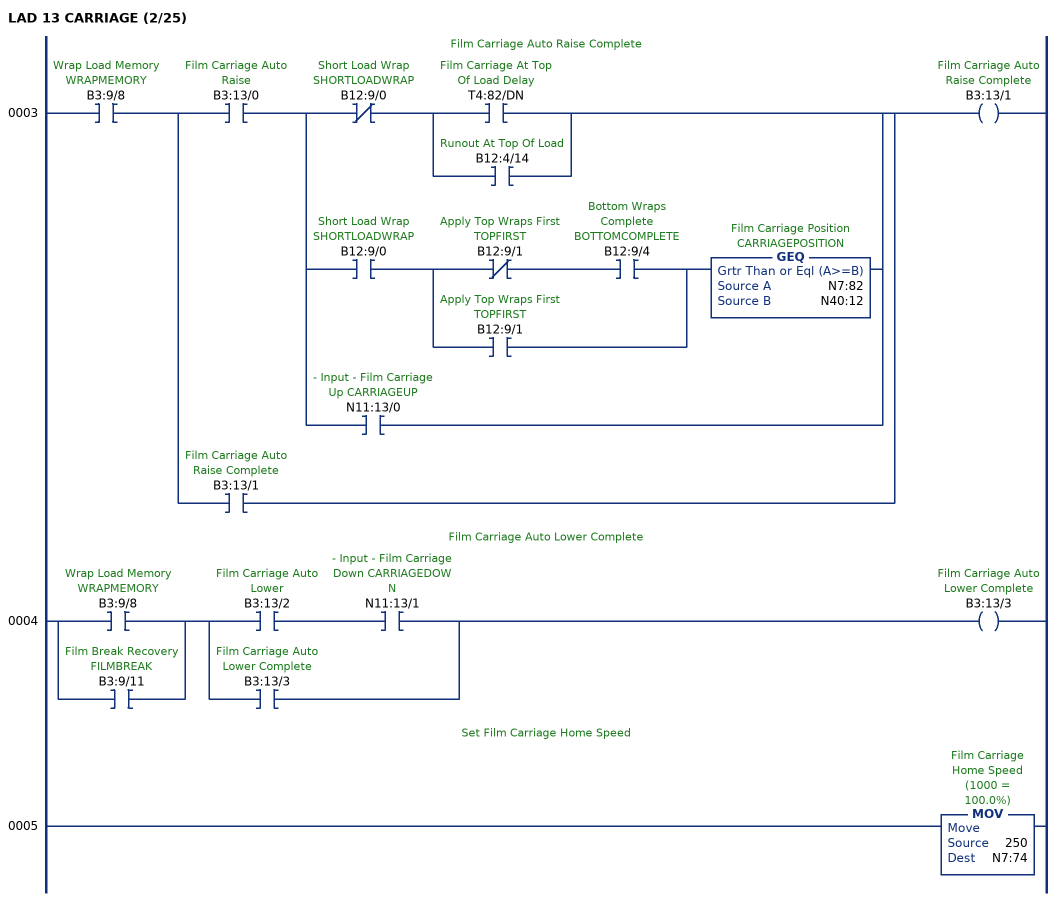
% Rung: 3 %
% Film Carriage Auto Raise Complete %
SOR XIC B3:9/8 BST XIC B3:13/0 BST XIO B12:9/0 BST XIC T4:82/DN NXB XIC B12:4/14 BND NXB XIC B12:9/0 BST XIO B12:9/1 XIC B12:9/4 NXB XIC B12:9/1 BND GEQ N7:82 N40:12 NXB XIC N11:13/0 BND NXB XIC B3:13/1 BND OTE B3:13/1 EOR
%   B3:9/8  WRAPMEMORY  "Wrap Load Memory" %
%   B3:13/0  "Film Carriage Auto Raise" %
%   B12:9/0  SHORTLOADWRAP  "Short Load Wrap" %
%   T4:82  "Film Carriage At Top Of Load Delay" %
%   B12:4/14  "Runout At Top Of Load" %
%   B12:9/1  TOPFIRST  "Apply Top Wraps First" %
%   B12:9/4  BOTTOMCOMPLETE  "Bottom Wraps Complete" %
%   N7:82  CARRIAGEPOSITION  "Film Carriage Position" %
%   N40:12  "Current Profile Short Load Height (Inches)" %
%   N11:13/0  CARRIAGEUP  "- Input - Film Carriage Up" %
%   B3:13/1  "Film Carriage Auto Raise Complete" %
% Rung: 4 %
% Film Carriage Auto Lower Complete %
SOR BST XIC B3:9/8 NXB XIC B3:9/11 BND BST XIC B3:13/2 XIC N11:13/1 NXB XIC B3:13/3 BND OTE B3:13/3 EOR
%   B3:9/8  WRAPMEMORY  "Wrap Load Memory" %
%   B3:9/11  FILMBREAK  "Film Break Recovery" %
%   B3:13/2  "Film Carriage Auto Lower" %
%   N11:13/1  CARRIAGEDOWN  "- Input - Film Carriage Down" %
%   B3:13/3  "Film Carriage Auto Lower Complete" %
% Rung: 5 %
% Set Film Carriage Home Speed %
SOR MOV 250 N7:74 EOR
%   N7:74  "Film Carriage Home Speed (1000 = 100.0%)" %

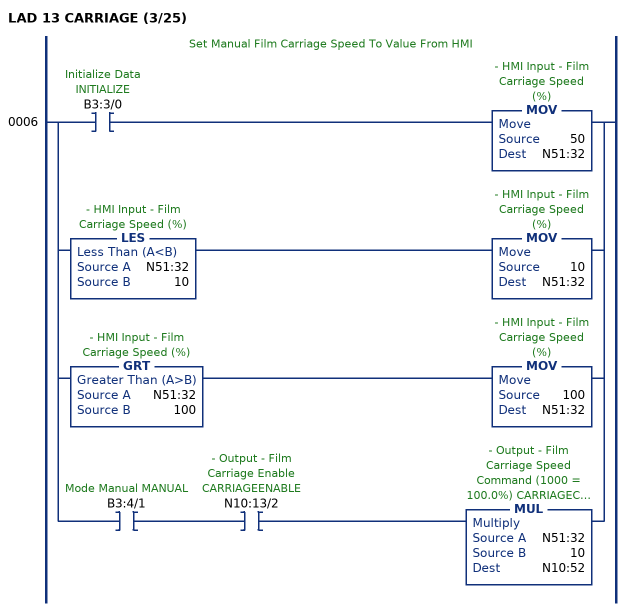
% Rung: 6 %
% Set Manual Film Carriage Speed To Value From HMI %
SOR BST BST XIC B3:3/0 MOV 50 N51:32 NXB LES N51:32 10 MOV 10 N51:32 NXB GRT N51:32 100 MOV 100 N51:32 BND NXB XIC B3:4/1 XIC N10:13/2 MUL N51:32 10 N10:52 BND EOR
%   B3:3/0  INITIALIZE  "Initialize Data" %
%   N51:32  "- HMI Input - Film Carriage Speed (%)" %
%   B3:4/1  MANUAL  "Mode Manual" %
%   N10:13/2  CARRIAGEENABLE  "- Output - Film Carriage Enable" %
%   N10:52  CARRIAGECOMMAND  "- Output - Film Carriage Speed Command (1000 = 100.0%)" %

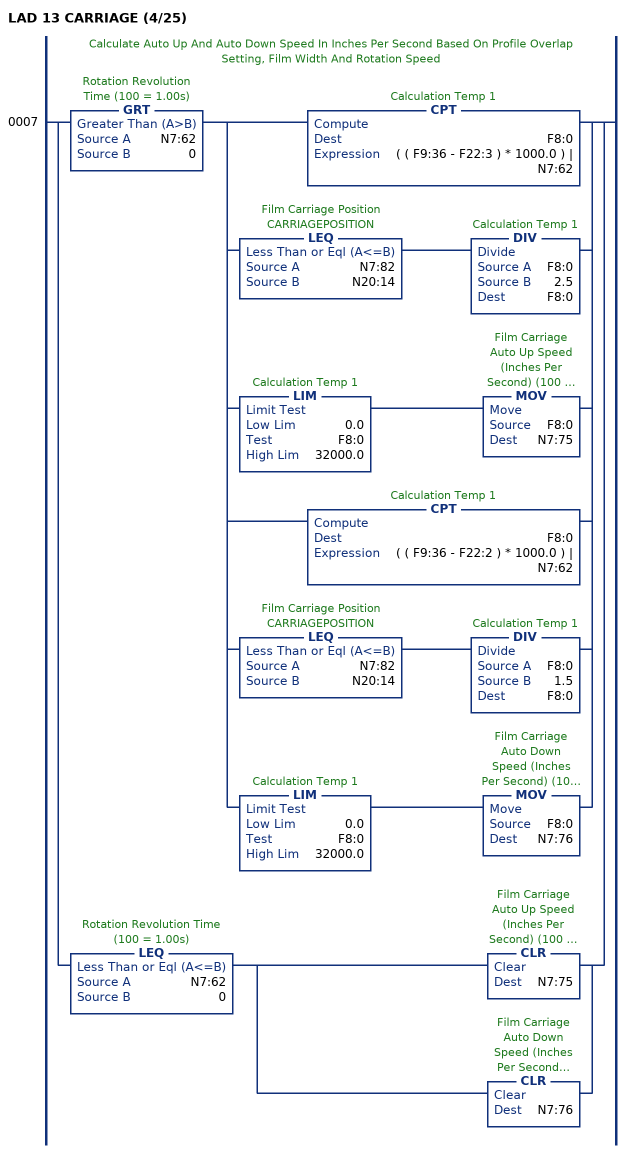
% Rung: 7 %
% Calculate Auto Up And Auto Down Speed In Inches Per Second Based On Profile Overlap Setting, Film Width And Rotation Speed %
SOR BST GRT N7:62 0 BST BST CPT F8:0 " ( ( F9:36 - F22:3 ) * 1000.0 ) | N7:62 " NXB LEQ N7:82 N20:14 DIV F8:0 2.5 F8:0 NXB LIM 0.0 F8:0 32000.0 MOV F8:0 N7:75 BND NXB BST CPT F8:0 " ( ( F9:36 - F22:2 ) * 1000.0 ) | N7:62 " NXB LEQ N7:82 N20:14 DIV F8:0 1.5 F8:0 NXB LIM 0.0 F8:0 32000.0 MOV F8:0 N7:76 BND BND NXB LEQ N7:62 0 BST CLR N7:75 NXB CLR N7:76 BND BND EOR
%   N7:62  "Rotation Revolution Time (100 = 1.00s)" %
%   F8:0  "Calculation Temp 1" %
%   F9:36  FILMWIDTHATLOAD  "Film Width At Load" %
%   F22:3  OVERLAPUP  "Overlap Up" %
%   N7:82  CARRIAGEPOSITION  "Film Carriage Position" %
%   N20:14  "Pallet-Grip Fully Released Position (10 = 10 Inches)" %
%   N7:75  "Film Carriage Auto Up Speed (Inches Per Second) (100 = 10.0 IPS)" %
%   F22:2  OVERLAPDOWN  "Overlap Down" %
%   N7:76  "Film Carriage Auto Down Speed (Inches Per Second) (100 = 10.0 IPS)" %

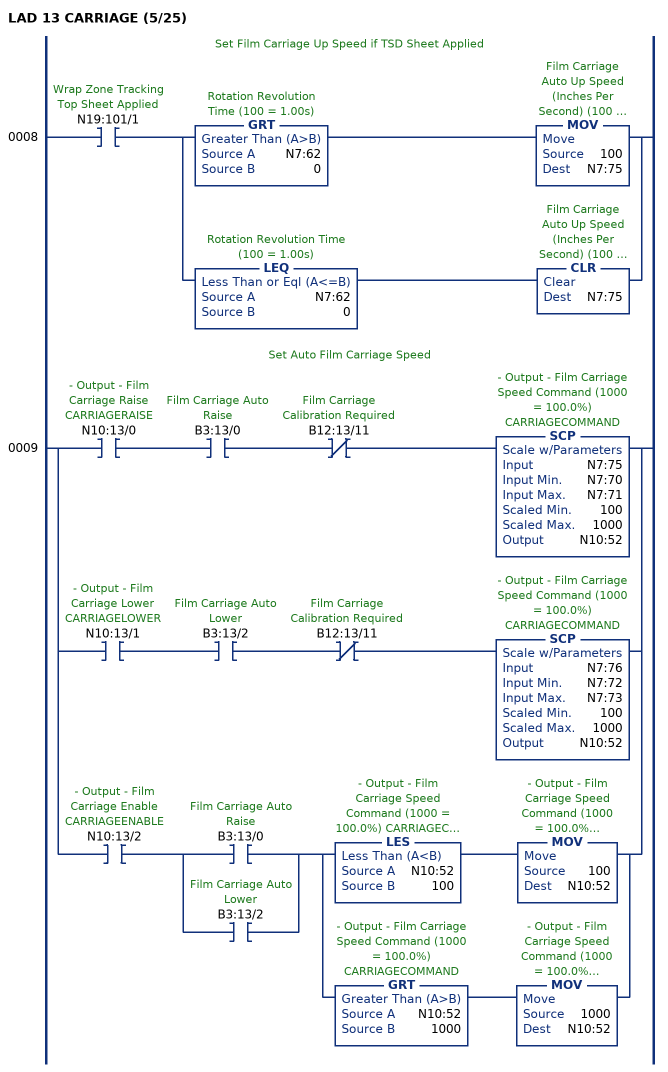
% Rung: 8 %
% Set Film Carriage Up Speed if TSD Sheet Applied %
SOR XIC N19:101/1 BST GRT N7:62 0 MOV 100 N7:75 NXB LEQ N7:62 0 CLR N7:75 BND EOR
%   N19:101/1  "Wrap Zone Tracking Top Sheet Applied" %
%   N7:62  "Rotation Revolution Time (100 = 1.00s)" %
%   N7:75  "Film Carriage Auto Up Speed (Inches Per Second) (100 = 10.0 IPS)" %
% Rung: 9 %
% Set Auto Film Carriage Speed %
SOR BST XIC N10:13/0 XIC B3:13/0 XIO B12:13/11 SCP N7:75 N7:70 N7:71 100 1000 N10:52 NXB XIC N10:13/1 XIC B3:13/2 XIO B12:13/11 SCP N7:76 N7:72 N7:73 100 1000 N10:52 NXB XIC N10:13/2 BST XIC B3:13/0 NXB XIC B3:13/2 BND BST LES N10:52 100 MOV 100 N10:52 NXB GRT N10:52 1000 MOV 1000 N10:52 BND BND EOR
%   N10:13/0  CARRIAGERAISE  "- Output - Film Carriage Raise" %
%   B3:13/0  "Film Carriage Auto Raise" %
%   B12:13/11  "Film Carriage Calibration Required" %
%   N7:75  "Film Carriage Auto Up Speed (Inches Per Second) (100 = 10.0 IPS)" %
%   N7:70  "Film Carriage Up Min Speed (Inches Per Second) (100 = 10.0 IPS)" %
%   N7:71  "Film Carriage Up Max Speed (Inches Per Second) (100 = 10.0 IPS)" %
%   N10:52  CARRIAGECOMMAND  "- Output - Film Carriage Speed Command (1000 = 100.0%)" %
%   N10:13/1  CARRIAGELOWER  "- Output - Film Carriage Lower" %
%   B3:13/2  "Film Carriage Auto Lower" %
%   N7:76  "Film Carriage Auto Down Speed (Inches Per Second) (100 = 10.0 IPS)" %
%   N7:72  "Film Carriage Down Min Speed (Inches Per Second) (100 = 10.0 IPS)" %
%   N7:73  "Film Carriage Down Max Speed (Inches Per Second) (100 = 10.0 IPS)" %
%   N10:13/2  CARRIAGEENABLE  "- Output - Film Carriage Enable" %

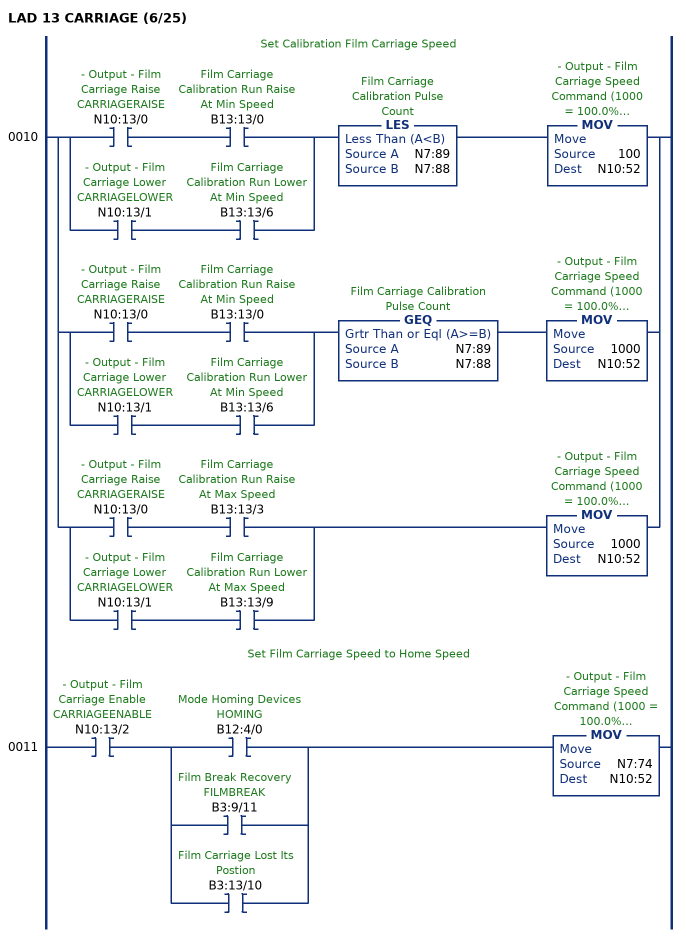
% Rung: 10 %
% Set Calibration Film Carriage Speed %
SOR BST BST XIC N10:13/0 XIC B13:13/0 NXB XIC N10:13/1 XIC B13:13/6 BND LES N7:89 N7:88 MOV 100 N10:52 NXB BST XIC N10:13/0 XIC B13:13/0 NXB XIC N10:13/1 XIC B13:13/6 BND GEQ N7:89 N7:88 MOV 1000 N10:52 NXB BST XIC N10:13/0 XIC B13:13/3 NXB XIC N10:13/1 XIC B13:13/9 BND MOV 1000 N10:52 BND EOR
%   N10:13/0  CARRIAGERAISE  "- Output - Film Carriage Raise" %
%   B13:13/0  "Film Carriage Calibration Run Raise At Min Speed" %
%   N10:13/1  CARRIAGELOWER  "- Output - Film Carriage Lower" %
%   B13:13/6  "Film Carriage Calibration Run Lower At Min Speed" %
%   N7:89  "Film Carriage Calibration Pulse Count" %
%   N7:88  "Film Carriage Speed Sample Preset" %
%   N10:52  CARRIAGECOMMAND  "- Output - Film Carriage Speed Command (1000 = 100.0%)" %
%   B13:13/3  "Film Carriage Calibration Run Raise At Max Speed" %
%   B13:13/9  "Film Carriage Calibration Run Lower At Max Speed" %
% Rung: 11 %
% Set Film Carriage Speed to Home Speed %
SOR XIC N10:13/2 BST XIC B12:4/0 NXB XIC B3:9/11 NXB XIC B3:13/10 BND MOV N7:74 N10:52 EOR
%   N10:13/2  CARRIAGEENABLE  "- Output - Film Carriage Enable" %
%   B12:4/0  HOMING  "Mode Homing Devices" %
%   B3:9/11  FILMBREAK  "Film Break Recovery" %
%   B3:13/10  "Film Carriage Lost Its Postion" %
%   N7:74  "Film Carriage Home Speed (1000 = 100.0%)" %
%   N10:52  CARRIAGECOMMAND  "- Output - Film Carriage Speed Command (1000 = 100.0%)" %

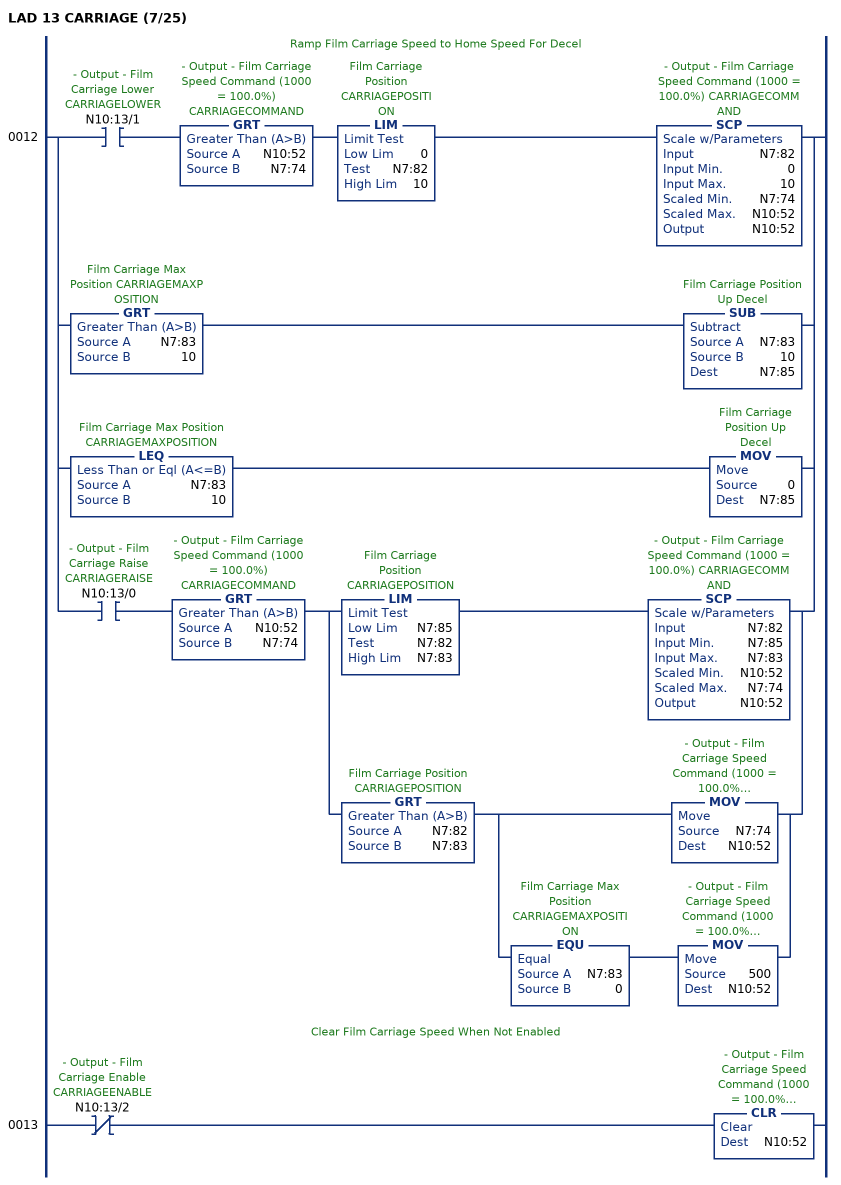
% Rung: 12 %
% Ramp Film Carriage Speed to Home Speed For Decel %
SOR BST XIC N10:13/1 GRT N10:52 N7:74 LIM 0 N7:82 10 SCP N7:82 0 10 N7:74 N10:52 N10:52 NXB BST GRT N7:83 10 SUB N7:83 10 N7:85 NXB LEQ N7:83 10 MOV 0 N7:85 BND NXB XIC N10:13/0 GRT N10:52 N7:74 BST LIM N7:85 N7:82 N7:83 SCP N7:82 N7:85 N7:83 N10:52 N7:74 N10:52 NXB GRT N7:82 N7:83 BST MOV N7:74 N10:52 NXB EQU N7:83 0 MOV 500 N10:52 BND BND BND EOR
%   N10:13/1  CARRIAGELOWER  "- Output - Film Carriage Lower" %
%   N10:52  CARRIAGECOMMAND  "- Output - Film Carriage Speed Command (1000 = 100.0%)" %
%   N7:74  "Film Carriage Home Speed (1000 = 100.0%)" %
%   N7:82  CARRIAGEPOSITION  "Film Carriage Position" %
%   N7:83  CARRIAGEMAXPOSITION  "Film Carriage Max Position" %
%   N7:85  "Film Carriage Position Up Decel" %
%   N10:13/0  CARRIAGERAISE  "- Output - Film Carriage Raise" %
% Rung: 13 %
% Clear Film Carriage Speed When Not Enabled %
SOR XIO N10:13/2 CLR N10:52 EOR
%   N10:13/2  CARRIAGEENABLE  "- Output - Film Carriage Enable" %
%   N10:52  CARRIAGECOMMAND  "- Output - Film Carriage Speed Command (1000 = 100.0%)" %

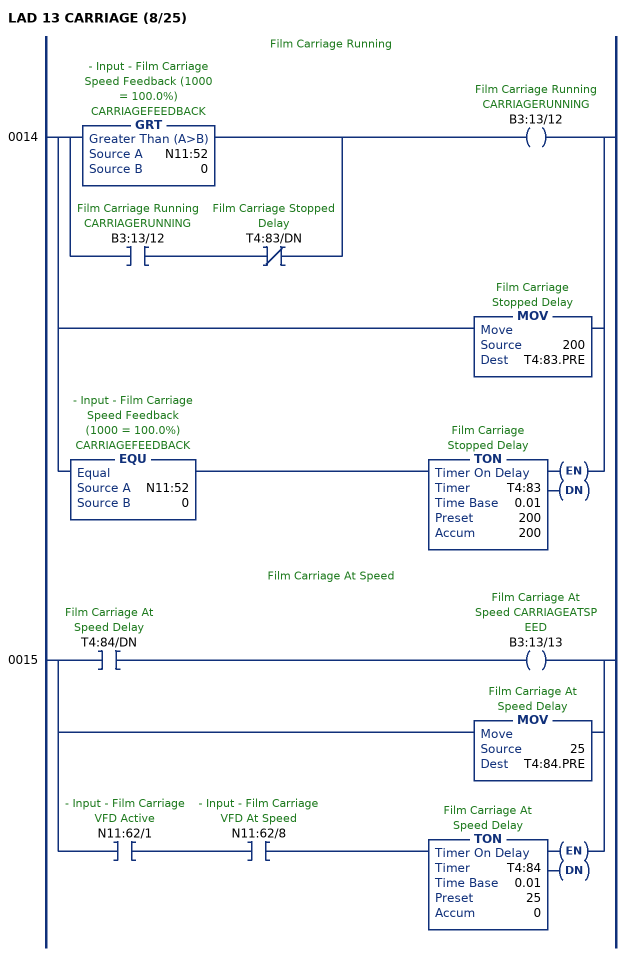
% Rung: 14 %
% Film Carriage Running %
SOR BST BST GRT N11:52 0 NXB XIC B3:13/12 XIO T4:83/DN BND OTE B3:13/12 NXB MOV 200 T4:83.PRE NXB EQU N11:52 0 TON T4:83 0.01 200 200 BND EOR
%   N11:52  CARRIAGEFEEDBACK  "- Input - Film Carriage Speed Feedback (1000 = 100.0%)" %
%   B3:13/12  CARRIAGERUNNING  "Film Carriage Running" %
%   T4:83  "Film Carriage Stopped Delay" %
% Rung: 15 %
% Film Carriage At Speed %
SOR BST XIC T4:84/DN OTE B3:13/13 NXB MOV 25 T4:84.PRE NXB XIC N11:62/1 XIC N11:62/8 TON T4:84 0.01 25 0 BND EOR
%   T4:84  "Film Carriage At Speed Delay" %
%   B3:13/13  CARRIAGEATSPEED  "Film Carriage At Speed" %
%   N11:62/1  "- Input - Film Carriage VFD Active" %
%   N11:62/8  "- Input - Film Carriage VFD At Speed" %

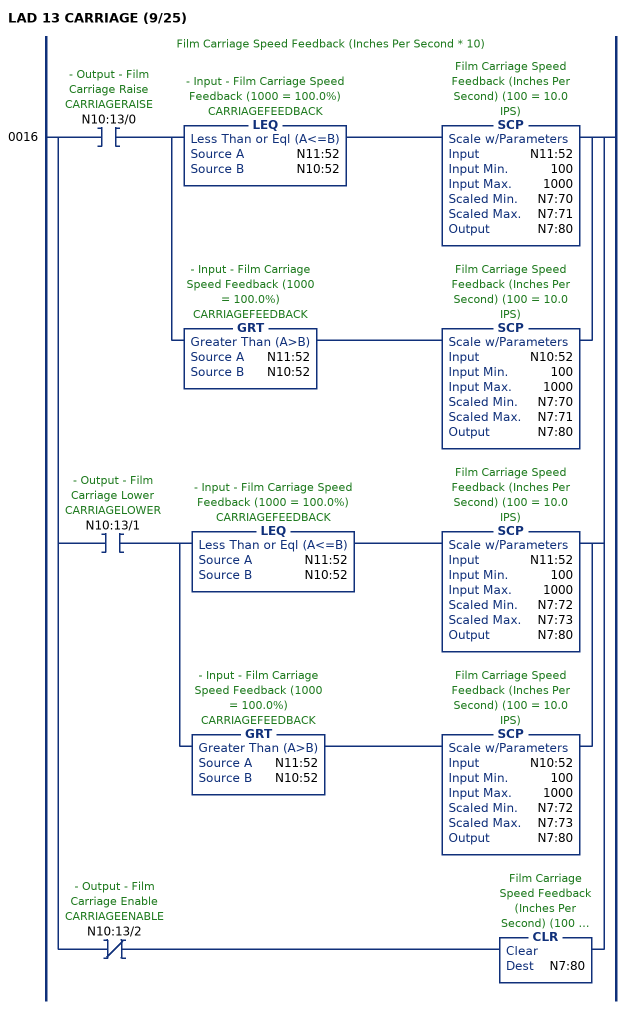
% Rung: 16 %
% Film Carriage Speed Feedback (Inches Per Second * 10) %
SOR BST XIC N10:13/0 BST LEQ N11:52 N10:52 SCP N11:52 100 1000 N7:70 N7:71 N7:80 NXB GRT N11:52 N10:52 SCP N10:52 100 1000 N7:70 N7:71 N7:80 BND NXB XIC N10:13/1 BST LEQ N11:52 N10:52 SCP N11:52 100 1000 N7:72 N7:73 N7:80 NXB GRT N11:52 N10:52 SCP N10:52 100 1000 N7:72 N7:73 N7:80 BND NXB XIO N10:13/2 CLR N7:80 BND EOR
%   N10:13/0  CARRIAGERAISE  "- Output - Film Carriage Raise" %
%   N11:52  CARRIAGEFEEDBACK  "- Input - Film Carriage Speed Feedback (1000 = 100.0%)" %
%   N10:52  CARRIAGECOMMAND  "- Output - Film Carriage Speed Command (1000 = 100.0%)" %
%   N7:70  "Film Carriage Up Min Speed (Inches Per Second) (100 = 10.0 IPS)" %
%   N7:71  "Film Carriage Up Max Speed (Inches Per Second) (100 = 10.0 IPS)" %
%   N7:80  "Film Carriage Speed Feedback (Inches Per Second) (100 = 10.0 IPS)" %
%   N10:13/1  CARRIAGELOWER  "- Output - Film Carriage Lower" %
%   N7:72  "Film Carriage Down Min Speed (Inches Per Second) (100 = 10.0 IPS)" %
%   N7:73  "Film Carriage Down Max Speed (Inches Per Second) (100 = 10.0 IPS)" %
%   N10:13/2  CARRIAGEENABLE  "- Output - Film Carriage Enable" %

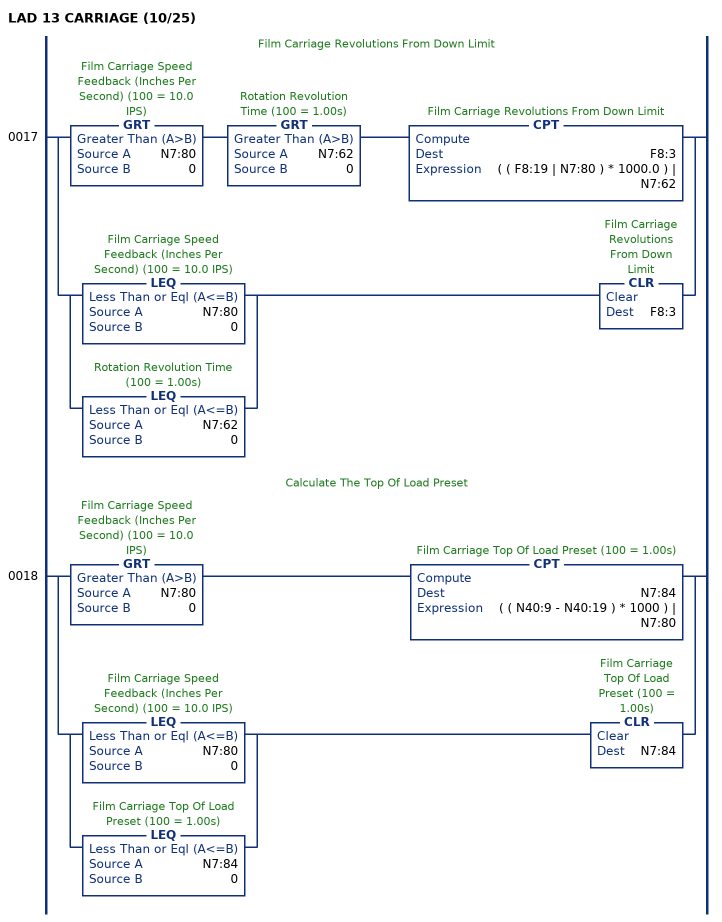
% Rung: 17 %
% Film Carriage Revolutions From Down Limit %
SOR BST GRT N7:80 0 GRT N7:62 0 CPT F8:3 " ( ( F8:19 | N7:80 ) * 1000.0 ) | N7:62 " NXB BST LEQ N7:80 0 NXB LEQ N7:62 0 BND CLR F8:3 BND EOR
%   N7:80  "Film Carriage Speed Feedback (Inches Per Second) (100 = 10.0 IPS)" %
%   N7:62  "Rotation Revolution Time (100 = 1.00s)" %
%   F8:3  "Film Carriage Revolutions From Down Limit" %
%   F8:19  "Film Carriage Position" %
% Rung: 18 %
% Calculate The Top Of Load Preset %
SOR BST GRT N7:80 0 CPT N7:84 " ( ( N40:9 - N40:19 ) * 1000 ) | N7:80 " NXB BST LEQ N7:80 0 NXB LEQ N7:84 0 BND CLR N7:84 BND EOR
%   N7:80  "Film Carriage Speed Feedback (Inches Per Second) (100 = 10.0 IPS)" %
%   N7:84  "Film Carriage Top Of Load Preset (100 = 1.00s)" %
%   N40:9  "Current Profile Top Overwrap (Inches)" %
%   N40:19  "Current Profile Top Overwrap Min Value (Inches)" %

